{attribute 'analysis' := '-33'}
PROGRAM INTERNAL PRG_MessageTests
VAR
    {IF defined (UNIT_TEST)}
    fbRoundTripMessageExampleTest : FB_RoundTripMessageExampleTest;
	
	// following tests using TcHaxx.Snappy.CLI (https://github.com/TcHaxx/snappy)
	fbScalarTypesTest	: FB_ScalarTypesTest;
	fbFooBarBazTests  	: FB_FooBarBazTests;
	fbComplexDataTests	: FB_ComplexDataTests;
	fbRepeatedComplexDataTests : FB_RepeatedComplexDataTests;
	fbMotorTests		: FB_MotorTests;
	fbDeviceTests 		: FB_DeviceTests;
    {END_IF}
END_VAR

END_PROGRAM

(* stored: Version 1.1.0.1
   POU PRG_MessageTests: Id {3a3ee01b-b87a-426e-9253-57e7b651cd6b}, SpecialFunc None *)
